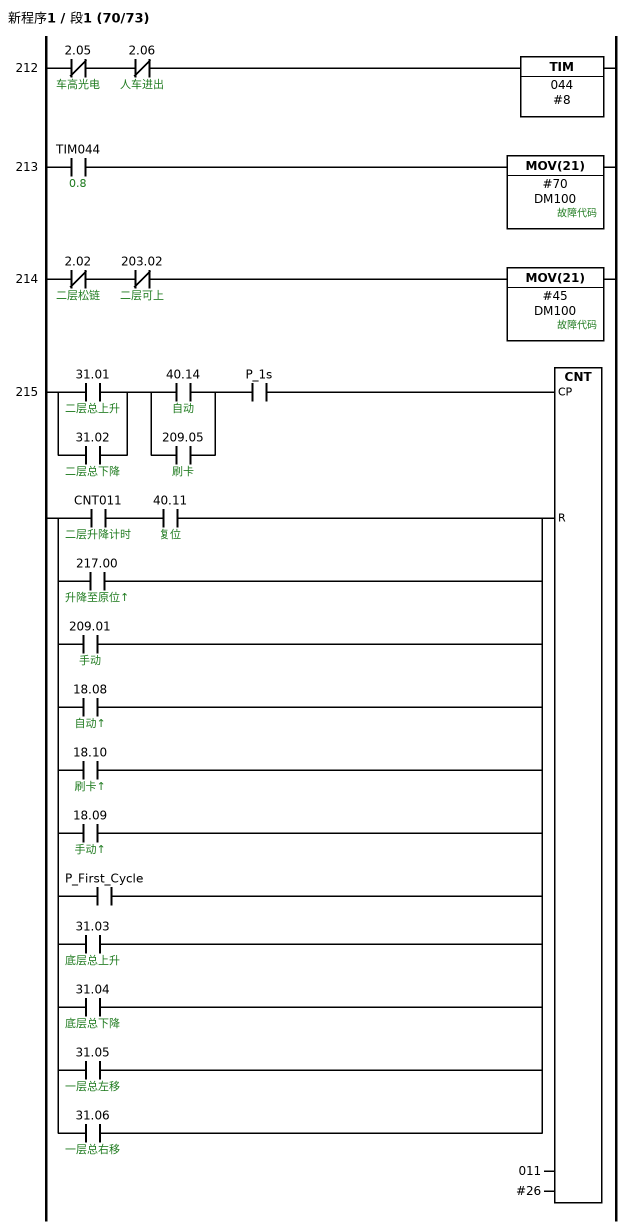
; [picture p72: 新程序1 / 段1, rungs 212-215]
; rung 212
LDNOT 2.05  ; 车高光电
ANDNOT 2.06  ; 人车进出
TIM 044 #8
; rung 213
LD TIM044  ; 0.8
MOV(21) #70 DM100  ; 故障代码
; rung 214
LDNOT 2.02  ; 二层松链
ANDNOT 203.02  ; 二层可上
MOV(21) #45 DM100  ; 故障代码
; rung 215
LD 31.01  ; 二层总上升
OR 31.02  ; 二层总下降
LD 40.14  ; 自动
OR 209.05  ; 刷卡
ANDLD
AND P_1s
LD CNT011  ; 二层升降计时
AND 40.11  ; 复位
OR 217.00  ; 升降至原位↑
OR 209.01  ; 手动
OR 18.08  ; 自动↑
OR 18.10  ; 刷卡↑
OR 18.09  ; 手动↑
OR P_First_Cycle
OR 31.03  ; 底层总上升
OR 31.04  ; 底层总下降
OR 31.05  ; 一层总左移
OR 31.06  ; 一层总右移
CNT 011 #26

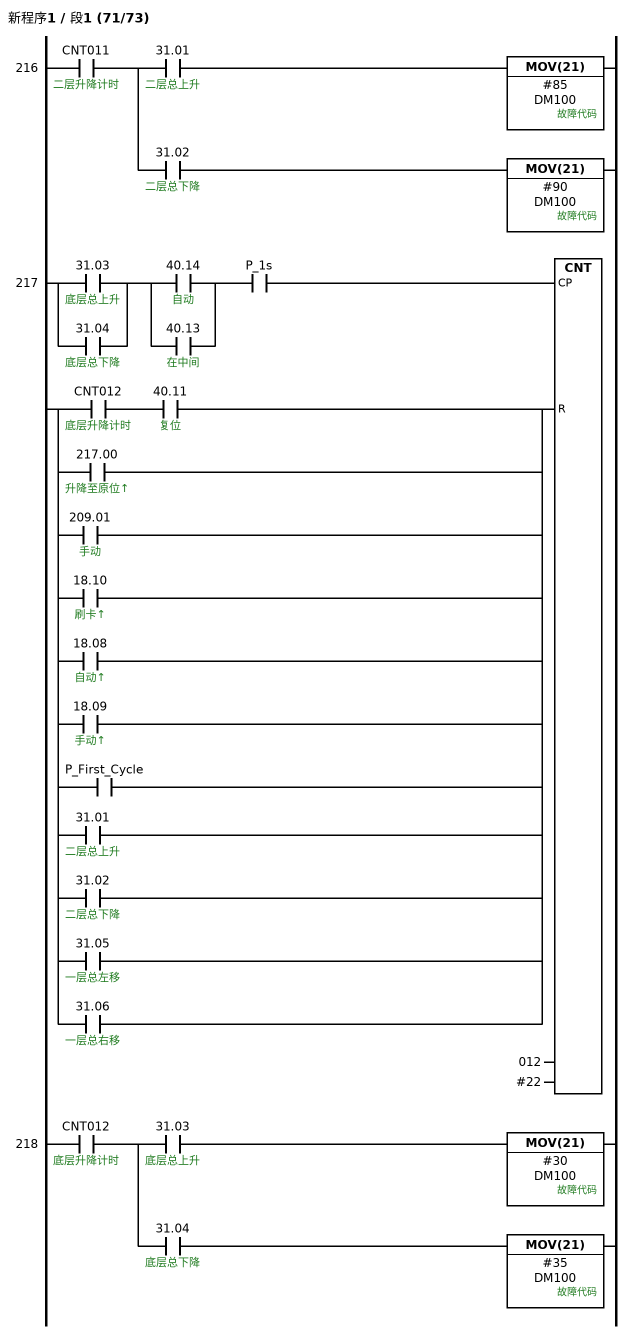
; rung 216
LD CNT011  ; 二层升降计时
OUT TR0
AND 31.01  ; 二层总上升
MOV(21) #85 DM100  ; 故障代码
LD TR0
AND 31.02  ; 二层总下降
MOV(21) #90 DM100  ; 故障代码
; rung 217
LD 31.03  ; 底层总上升
OR 31.04  ; 底层总下降
LD 40.14  ; 自动
OR 40.13  ; 在中间
ANDLD
AND P_1s
LD CNT012  ; 底层升降计时
AND 40.11  ; 复位
OR 217.00  ; 升降至原位↑
OR 209.01  ; 手动
OR 18.10  ; 刷卡↑
OR 18.08  ; 自动↑
OR 18.09  ; 手动↑
OR P_First_Cycle
OR 31.01  ; 二层总上升
OR 31.02  ; 二层总下降
OR 31.05  ; 一层总左移
OR 31.06  ; 一层总右移
CNT 012 #22
; rung 218
LD CNT012  ; 底层升降计时
OUT TR0
AND 31.03  ; 底层总上升
MOV(21) #30 DM100  ; 故障代码
LD TR0
AND 31.04  ; 底层总下降
MOV(21) #35 DM100  ; 故障代码

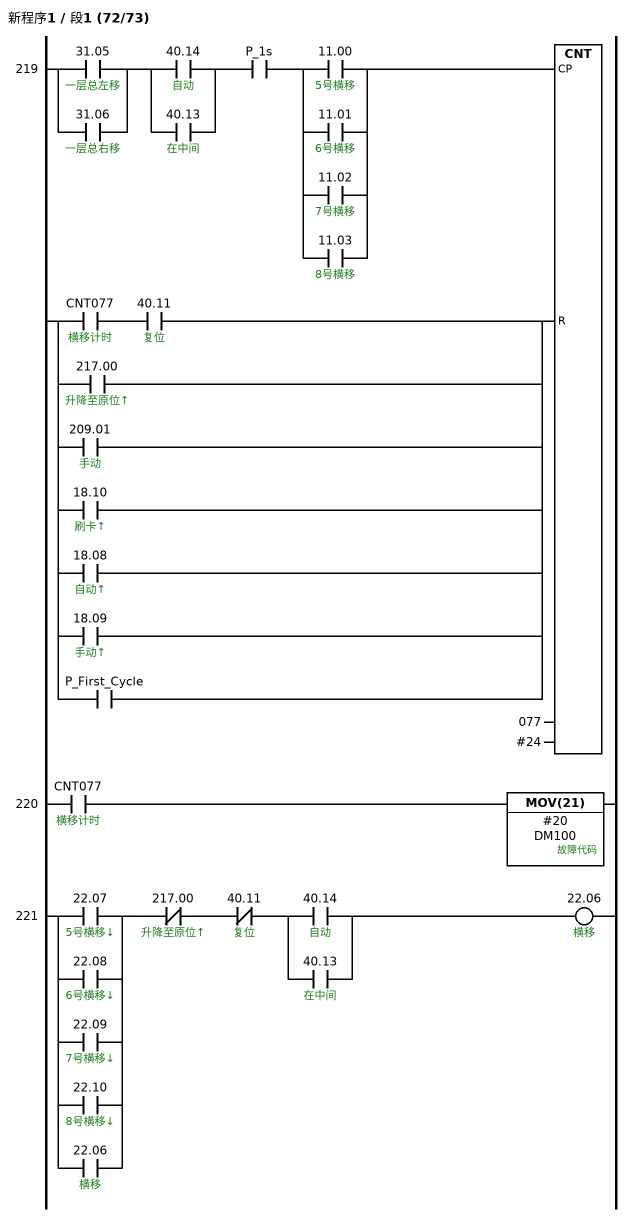
; rung 219
LD 31.05  ; 一层总左移
OR 31.06  ; 一层总右移
LD 40.14  ; 自动
OR 40.13  ; 在中间
ANDLD
AND P_1s
LD 11.00  ; 5号横移
OR 11.01  ; 6号横移
OR 11.02  ; 7号横移
OR 11.03  ; 8号横移
ANDLD
LD CNT077  ; 横移计时
AND 40.11  ; 复位
OR 217.00  ; 升降至原位↑
OR 209.01  ; 手动
OR 18.10  ; 刷卡↑
OR 18.08  ; 自动↑
OR 18.09  ; 手动↑
OR P_First_Cycle
CNT 077 #24
; rung 220
LD CNT077  ; 横移计时
MOV(21) #20 DM100  ; 故障代码
; rung 221
LD 22.07  ; 5号横移↓
OR 22.08  ; 6号横移↓
OR 22.09  ; 7号横移↓
OR 22.10  ; 8号横移↓
OR 22.06  ; 横移
ANDNOT 217.00  ; 升降至原位↑
ANDNOT 40.11  ; 复位
LD 40.14  ; 自动
OR 40.13  ; 在中间
ANDLD
OUT 22.06  ; 横移

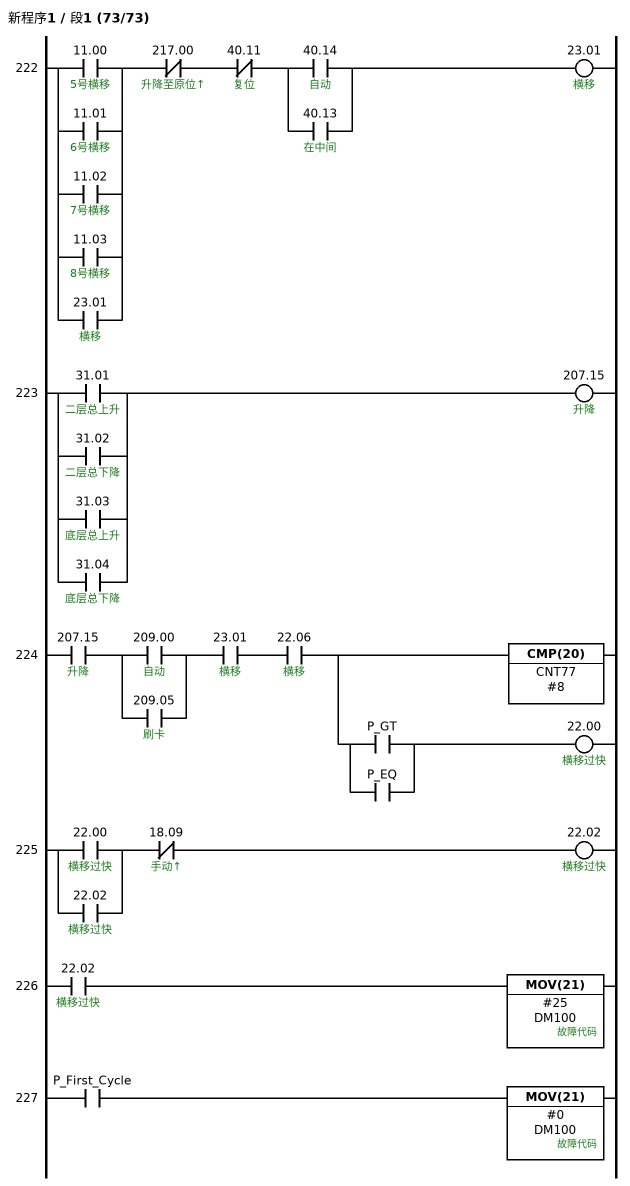
; rung 222
LD 11.00  ; 5号横移
OR 11.01  ; 6号横移
OR 11.02  ; 7号横移
OR 11.03  ; 8号横移
OR 23.01  ; 横移
ANDNOT 217.00  ; 升降至原位↑
ANDNOT 40.11  ; 复位
LD 40.14  ; 自动
OR 40.13  ; 在中间
ANDLD
OUT 23.01  ; 横移
; rung 223
LD 31.01  ; 二层总上升
OR 31.02  ; 二层总下降
OR 31.03  ; 底层总上升
OR 31.04  ; 底层总下降
OUT 207.15  ; 升降
; rung 224
LD 207.15  ; 升降
LD 209.00  ; 自动
OR 209.05  ; 刷卡
ANDLD
AND 23.01  ; 横移
AND 22.06  ; 横移
CMP(20) CNT77 #8
LD P_GT
OR P_EQ
ANDLD
OUT 22.00  ; 横移过快
; rung 225
LD 22.00  ; 横移过快
OR 22.02  ; 横移过快
ANDNOT 18.09  ; 手动↑
OUT 22.02  ; 横移过快
; rung 226
LD 22.02  ; 横移过快
MOV(21) #25 DM100  ; 故障代码
; rung 227
LD P_First_Cycle
MOV(21) #0 DM100  ; 故障代码
; rung 228
END(01)